//FB sends a "command" out and waits for response of the connected device (handshake mode)
//By setting pDest = 0 the FB will turn into only send mode and with pSrc = 0 into only receive mode (ClrComBuffer will be ignored)
FUNCTION_BLOCK ComPortDeviceCom_SendRecBytes
VAR CONSTANT
	TIMEOUT_COM												: TIME 		:= T#10S;
END_VAR
VAR_INPUT
	Execute													: BOOL;
	ClrComBuffer											: BOOL := TRUE; //TRUE Clears com buffer before start
	Prefix													: STRING(5) := ''; //Use string variable as byte array if Prefix is not a string
	Suffix													: STRING(5) := '$r$n'; //Use string variable as byte array if Suffix is not a string
	RecTimeout												: TIME := DEFAULT_ADS_TIMEOUT; 
	pSrc													: POINTER TO BYTE; //Pointer to data source, in case the pointer is empty (0) the FB will only start to wait for data
	cbSrcLen												: UDINT;
	pDest													: POINTER TO BYTE; //Pointer to receive buffer, in case the pointer is empty (0) the FB will send data out 
	cbDestLen												: UDINT;
END_VAR
VAR_IN_OUT
	Handle													:	ComPortDeviceCom_BufferHandle;
END_VAR	
VAR_OUTPUT
	RecBytes												: UDINT;	
	Done													: BOOL;
	Busy													: BOOL;
	Error													: BOOL;
	ErrorID													: ComError_t := ComError_t.COMERROR_NOERROR;
END_VAR
VAR
(* Memory *****************************************************)
	state													: INT := 0;
	
(* Timer ******************************************************)
	timeout													:	ton := (PT := TIMEOUT_COM);
	
(* Trigger ****************************************************)
	rtExecute												: R_TRIG;
	
(* Blocks *****************************************************)
	Rec														: ReceiveData := (Timeout := T#10S);
	Send													: SendData;
	
(* Error ******************************************************)
(* Dummys *****************************************************)
END_VAR

	(* Send data and receive response						 *)
	(*********************************************************)
	
(* state machine ********************************************************)
	rtExecute(CLK := Execute);
	CASE state OF
	0 : 
		Busy 												:= FALSE;
		IF NOT Execute THEN
			Done 											:= FALSE;
			Error 											:= FALSE;
			ErrorID 										:= 0;
		END_IF
		IF rtExecute.Q THEN
			Busy 											:= TRUE;		
			timeout(IN := FALSE, PT := TIMEOUT_COM + RecTimeout);
			RecBytes 										:= 0;
			Error 											:= FALSE;
			ErrorID 										:= ComError_t.COMERROR_NOERROR;
			Rec(Reset := TRUE,Timeout :=RecTimeout,rxBuffer := Handle.RXBuffer);	
		
			IF ClrComBuffer
			THEN
				Handle.Clear();
			END_IF
			
			IF pSrc = 0 AND pDest <> 0
			THEN //Rec mode
				MemSet(pDest,0,cbDestLen);
				Rec(
					Reset := FALSE,
					pPrefix:= SEL(Prefix[0] > 0, 0, ADR(Prefix)), pSuffix:= SEL(Suffix[0] > 0, 0, ADR(Suffix)), 
					LenPrefix := TO_BYTE(LEN(Prefix)), LenSuffix := TO_BYTE(LEN(Suffix)),					
					pReceiveData:= pDest, SizeReceiveData:= cbDestLen, 
					rxBuffer := Handle.RXBuffer);
				state 										:= 2;	
			ELSE
				Send(pSendData := pSrc, Length := cbSrcLen,TxBuffer := handle.TXBuffer);
				state 										:= state + 1;			
			END_IF
		END_IF
		
	1 : //Send tag 
		IF Send.Busy  //Call FB only if still busy after call in state 0
		THEN
			Send(pSendData := pSrc, Length := cbSrcLen,TxBuffer := handle.TXBuffer);
		END_IF
		IF NOT Send.Busy 
		THEN
			IF Send.Error <> ComError_t.COMERROR_NOERROR
			THEN
				Busy										:= FALSE;
				Error										:= TRUE;
				Errorid										:= Send.Error;
				state										:= 0;
			ELSIF pDest = 0
			THEN
				Busy										:= FALSE;
				Done										:= TRUE;
				state										:= 0;			
			ELSE
				MemSet(pDest,0,cbDestLen);
				Rec(
					Reset := FALSE,
					pPrefix:= SEL(Prefix[0] > 0, 0, ADR(Prefix)), pSuffix:= SEL(Suffix[0] > 0, 0, ADR(Suffix)), 
					LenPrefix := TO_BYTE(LEN(Prefix)), LenSuffix := TO_BYTE(LEN(Suffix)),					
					pReceiveData:= pDest, SizeReceiveData:= cbDestLen, 
					rxBuffer := Handle.RXBuffer);
				
				state 										:= state + 1;
			END_IF
		END_IF

	2: //Wair for response
		timeout(IN := TRUE);
		Rec(
			pPrefix:= SEL(Prefix[0] > 0, 0, ADR(Prefix)), pSuffix:= SEL(Suffix[0] > 0, 0, ADR(Suffix)), 
			LenPrefix := TO_BYTE(LEN(Prefix)), LenSuffix := TO_BYTE(LEN(Suffix)),	
			pReceiveData:= pDest, SizeReceiveData:= cbDestLen, 
			rxBuffer := Handle.RXBuffer);
		IF NOT Rec.Busy
		THEN
			IF Rec.DataReceived
			THEN
				IF Rec.LenReceiveData > 0
				THEN
					RecBytes								:= Rec.LenReceiveData;					
					Busy									:= FALSE;
					Done									:= TRUE;
					state									:= 0;					
				ELSE
					; //Nothing received, continue to read until done or timeout kicks in
				END_IF
			ELSIF Rec.Error <> ComError_t.COMERROR_NOERROR
			THEN
				Busy										:= FALSE;
				Error										:= TRUE;
				Errorid										:= Rec.Error;
				state										:= 0;								
			ELSIF Rec.RxTimeout 
			THEN
				Busy										:= FALSE;
				Error										:= TRUE;
				Errorid										:= ComError_t.COMERROR_TIMEOUT;
				state										:= 0;	
			ELSIF timeout.Q
			THEN
				Busy										:= FALSE;
				Error										:= TRUE;
				Errorid										:= ComError_t.COMERROR_TIMEOUT;
				state										:= 0;					
			END_IF
		END_IF
	END_CASE
(********************************************************************************)

END_FUNCTION_BLOCK

(* stored: Version 1.1.0.1, ProductVersion 3.1.4024.13
   POU ComPortDeviceCom_SendRecBytes: Id {2b2e6a6b-90e8-4fdd-8fd3-b70dc45690aa}, SpecialFunc None *)
